{attribute 'qualified_only'}
VAR_GLOBAL
	
	enableAxi: ARRAY[1..10] OF BOOL;
	runFWD: ARRAY[1..10] OF BOOL;
	resetAxi: ARRAY[1..10] OF BOOL;
	revs: REAL;
	mL_target: REAL;
	runBWD: ARRAY[1..10] OF BOOL;
	enableValv: ARRAY[1..5] OF BOOL;
	valvPos: INT;
	calibResult: ARRAY[1..50] OF ST_Results;
	
END_VAR

(* stored: Version 1.1.0.1, ProductVersion 3.1.4024.15
   GVL GVL_Marco: Id {80397fe9-0a64-47cf-a8bc-5c0cd05c5f13} *)
